{attribute 'qualified_only'}
VAR_GLOBAL
    nAssertFailuresCount : UINT;
    nAssertSuccessCount : UINT;
END_VAR

(* stored: Version 1.1.0.1, ProductVersion 3.1.4022.12
   GVL GVL_AssertResult: Id {e58ca29c-1ff3-4ff2-ac0d-06192d9ad9fb} *)
